SUBAPPLICATION Uebung_021 (* Spiegelabfolge (1) *)
  (* Standard: 61499-2; Description: Copyright (c) 2023 Meisterschulen am Ostbahnhof This program and the accompanying materials are made available under the terms of the Eclipse Public License 2.0 which is available at https://www.eclipse.org/legal/epl-2.0/ SPDX-License-Identifier: EPL-2.0 *)
  (* Version 1.0, 2023-10-23, Franz Höpfinger, Meisterschulen am Ostbahnhof *)
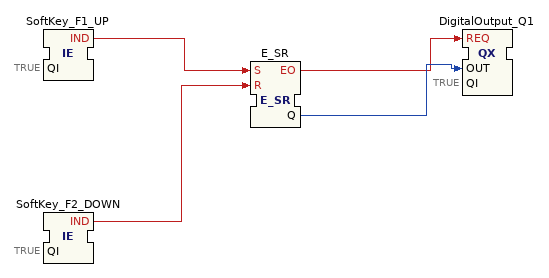
  (* START-Knopf *)
  (* Endlage *)
  FBS
    DigitalOutput_Q1 : QX(QI := TRUE);
    SoftKey_F1_UP : IE(QI := TRUE);
    E_SR : E_SR;
    SoftKey_F2_DOWN : IE(QI := TRUE);
  END_FBS
  EVENT_CONNECTIONS
    SoftKey_F1_UP.IND TO E_SR.S;
    SoftKey_F2_DOWN.IND TO E_SR.R;
    E_SR.EO TO DigitalOutput_Q1.REQ;
  END_CONNECTIONS
  DATA_CONNECTIONS
    E_SR.Q TO DigitalOutput_Q1.OUT;
  END_CONNECTIONS
END_SUBAPPLICATION
